// TIA Portal V20 export
VAR_GLOBAL   // PLC tag table "Default tag table_4"
   sensor AT %I0.0 : Bool;
END_VAR
